FUNCTION_BLOCK Pulser
VAR_INPUT
	// Width of the counted ON pulse
	ShortPulseWidth : TIME := T#200MS;
	// Width of the paused ON pulse
	LongPulseWidth : TIME := T#2S;
	// Width of the deadtime between pulses
	DeadPulseWidth : TIME := T#300MS;
END_VAR
VAR_OUTPUT
END_VAR
VAR
END_VAR

METHOD M_Pulse : BOOL
VAR_INPUT
	// If the pulsing should be ON or OFF if OFF the return value will also be LOW/OFF
	Active : BOOL;
	// Number of short pulses
	Pulses : INT := 0;
END_VAR
VAR_INST
	pulseCounter : INT := 0;
	state : INT := 0;
	timer : TP;
END_VAR

// Return immediatly if not active.
IF NOT Active THEN
	pulseCounter := 0;
	M_Pulse := FALSE;
	state := 0;
	timer(IN:=FALSE);
	RETURN;
END_IF

// special case if 0 pulses are requested
IF Pulses <= 0 THEN
	pulseCounter := 0;
	M_Pulse := TRUE;
	state := 0;
	timer(IN:=FALSE);
	RETURN;
END_IF


CASE state OF
0: // Start the timer for high signal
	M_Pulse := TRUE;
	timer(IN:=TRUE,PT:=LongPulseWidth);
	state := 1;
1: // alive time
	IF timer.Q THEN // Keep high
		M_Pulse := TRUE;
		timer(IN:=FALSE);
	ELSE // start timer for low periode
		M_Pulse := FALSE;
		timer(IN:=TRUE,PT:=DeadPulseWidth);
		state := 2;		
	END_IF
2: // deadtime
	IF timer.Q THEN // keep low
		M_Pulse := FALSE;
		timer(IN:=FALSE);
	ELSE // start timer for high periode
		M_Pulse := TRUE;
		pulseCounter := pulseCounter + 1;
		IF pulseCounter >= Pulses THEN
			pulseCounter := 0;
			timer(IN:=TRUE,PT:=LongPulseWidth);
		ELSE
			timer(IN:=TRUE,PT:=ShortPulseWidth);
		END_IF
		state := 1;		
	END_IF
END_CASE
END_METHOD

END_FUNCTION_BLOCK

(* stored: Version 1.1.0.1, ProductVersion 3.1.4024.10
   POU Pulser: Id {4496ebad-26b5-422d-9b61-9c396183ec0a}, SpecialFunc None
   Method M_Pulse: Id {3ee845d1-4402-41df-9bb0-d436d4c2d2b9} *)
